PROGRAM test_vacuum

VAR
	Vacuum_post1:REAL;
	Vacuum_post2:REAL;
	Vacuum_post3:REAL;
	Vacuum_post4:REAL;

END_VAR



Vacuum_post1:= ((Vacuum_Station1 - 8.0)* 3.8/16.0/2000)-1;
Vacuum_post2:= ((Vacuum_Station2 - 8.0)* 4.0/16.0/2000)-1;
Vacuum_post3:= ((Vacuum_Station3 - 8.0)* 4.0/16.0/2000)-1;
Vacuum_post4:= ((Vacuum_Station4 - 8.0)* 4.0/16.0/2000)-1;

END_PROGRAM

(* stored: Version 1.1.0.1, ProductVersion 3.1.0.26
   POU test_vacuum: Id {aef989de-6a1d-444b-9105-4f22692472fc} *)
